{attribute 'linkalways'} 
{attribute 'no_explicit_call' := 'This FB is a CLASS and must be accessed using methods or properties'}
{attribute 'enable_dynamic_creation'}
FUNCTION_BLOCK ABSTRACT JsonDeserializerEvent EXTENDS Disposable
VAR
	_target : I_JsonDeserializer;
END_VAR

METHOD FB_init : BOOL
VAR_INPUT
	bInitRetains : BOOL; // if TRUE, the retain variables are initialized (warm start / cold start)
	bInCopyCode : BOOL;  // if TRUE, the instance afterwards gets moved into the copy code (online change)
	Target : I_JsonDeserializer;
END_VAR
This^._target := Target;
END_METHOD

PROPERTY PUBLIC Target : I_JsonDeserializer
GET // PUBLIC
Target := _target;
END_GET
END_PROPERTY

END_FUNCTION_BLOCK

(* stored: Version 1.1.0.1, ProductVersion 3.1.4024.12
   POU JsonDeserializerEvent: Id {278df70c-9a81-48a4-8a48-b438945815cb}, SpecialFunc None
   Folder Constructor: Id {3ba864cc-74c4-4416-9bc6-62780b499fcb}
   Method FB_init: Id {dba50271-a49a-4367-a25f-dd6776786a0b}
   Property Target: Id {cac5726d-a4f9-4aa5-af6f-109d0275f5f8}
   Get Get: Id {16dfc4ea-9f84-4845-8ac7-c14c0627e8fc} *)
